(* CODESYS project tcl_stringutils.library
   Company: Red Rock Controls Limited
   Description: F_String_To_IPv4_Address added
   Version: 1.1.3.0
   Placeholder: tcl_StringUtils
   Author: Roger Christopher
   Title: tcl_StringUtils

Project tree, tasks and I/O mapping:
  libraries: Tc2_Standard, * (Beckhoff Automation GmbH); Tc2_System, * (Beckhoff Automation GmbH); Tc2_Utilities, * (Beckhoff Automation GmbH); Tc3_Module, * (Beckhoff Automation GmbH)
  Classes/
    function block T_LongString [ST]: AppendString, Clear, Address, Length
    function block T_StringSplitter [ST]: GetNext, GetRemainder, HasMore, Init
  Functions/
    Conversion/
      function F_String_To_IPv4_Address [ST]
      function F_TypeClassToString [ST]
      function F_ULINT_TO_TIMESTRUCT [ST]
    Date Time Formatting/
      function F_DateAsString [ST]
      function F_DateTimeAsString [ST]
      function F_DateTimeAsString_ms [ST]
      function F_TimeAsString [ST]
      function F_TimeAsString_ms [ST]
      function F_TimestampAsFilenameString [ST]
    String Formatting/
      function F_FormatString1 [ST]
      function F_FormatString10 [ST]
      function F_FormatString2 [ST]
      function F_FormatString3 [ST]
      function F_FormatString4 [ST]
      function F_FormatString5 [ST]
      function F_FormatString6 [ST]
      function F_FormatString7 [ST]
      function F_FormatString8 [ST]
      function F_FormatStringEx1 [ST]
      function F_FormatStringEx10 [ST]
      function F_FormatStringEx2 [ST]
      function F_FormatStringEx3 [ST]
      function F_FormatStringEx4 [ST]
      function F_FormatStringEx5 [ST]
      function F_FormatStringEx6 [ST]
      function F_FormatStringEx7 [ST]
      function F_FormatStringEx8 [ST]
      function F_LREAL_TO_STRING [ST]
      function F_LTrimEx [ST]
      function F_PadString [ST]
      function F_RTrimEx [ST]
      function F_STRING_TO_ARG [ST]
      function F_Trim [ST]
  Version/
    global variables Global_Version
  text list GlobalTextList
  global variables Param
*)

// Version/Global_Version
{attribute 'TcGenerated'}
{attribute 'no-analysis'}
{attribute 'linkalways'}
// This function has been automatically generated from the project information.
VAR_GLOBAL CONSTANT
	{attribute 'const_non_replaced'}
	stLibVersion_tcl_StringUtils : ST_LibVersion := (iMajor := 1, iMinor := 1, iBuild := 3, iRevision := 0, nFlags := 0, sVersion := '1.1.3.0');
END_VAR

// Param
{attribute 'qualified_only'}
VAR_GLOBAL CONSTANT
    MaxCsvFields : INT := 99;
END_VAR

// Classes/T_LongString
FUNCTION_BLOCK T_LongString
VAR
    buffer : STRING(MAX_LENGTH);
    CharCount : UDINT;
END_VAR
VAR CONSTANT
    MAX_LENGTH : UDINT := 1024;
END_VAR

METHOD AppendString
VAR_INPUT
    str : T_MaxString;
END_VAR
VAR
    stringLength : UDINT;
END_VAR
stringLength := INT_TO_UDINT(LEN(str));

IF (stringLength + CharCount < MAX_LENGTH - 1) THEN
    MEMCPY(
        destAddr := Address + CharCount,
        srcAddr  := ADR(str),
        n        := stringLength);
    CharCount := CharCount + stringLength;       
END_IF
END_METHOD

METHOD Clear
VAR_INPUT
END_VAR
MEMSET(Address,0,MAX_LENGTH);
CharCount := 0;
END_METHOD

PROPERTY Address : PVOID
GET
Address := ADR(Buffer);
END_GET
END_PROPERTY

PROPERTY Length : UDINT
GET
Length := CharCount;
END_GET
END_PROPERTY

END_FUNCTION_BLOCK

// Classes/T_StringSplitter
FUNCTION_BLOCK T_StringSplitter
VAR
	SubjectString : TC2_SYSTEM.T_MaxString;
	Delimiter : STRING;
	Delimiter1 : STRING;
	Delimiter2 : STRING;
	NextDelimiterPosition : INT;
	NextDelimiter1Position : INT;
	NextDelimiter2Position : INT;
END_VAR

METHOD GetNext : STRING(255)
VAR_INPUT
END_VAR
VAR
	RemainingLength: INT;
END_VAR
NextDelimiter1Position := FIND(SubjectString , Delimiter1);
NextDelimiter2Position := FIND(SubjectString , Delimiter2);

IF NextDelimiter1Position = 0 THEN
    // use Delimiter 2 position , even if zero...
    NextDelimiterPosition := NextDelimiter2Position;
    Delimiter := Delimiter2;
    
ELSIF NextDelimiter2Position = 0 THEN
    // use Delimiter 1 position , non-zero...
    NextDelimiterPosition := NextDelimiter1Position;
    Delimiter := Delimiter1;

ELSE
    // Both delimters found - use the one nearest the start of the string...
    IF NextDelimiter1Position < NextDelimiter2Position THEN
        NextDelimiterPosition := NextDelimiter1Position;
        Delimiter := Delimiter1;
    ELSE
        NextDelimiterPosition := NextDelimiter2Position;
        Delimiter := Delimiter2;
	END_IF
END_IF

IF NextDelimiterPosition > 0 THEN // delimitter found
    
    // extract next sub-string
	GetNext := LEFT(SubjectString,NextDelimiterPosition - 1);
    
    // remove sub-string from subject string
	RemainingLength := LEN(SubjectString) - NextDelimiterPosition - LEN(Delimiter) + 1;
	SubjectString := RIGHT(SubjectString,RemainingLength);
    
//    // strip any delimitters from front of remaining string
//    WHILE FIND(SubjectString,Delimiter1) = 1 DO
//        SubjectString := RIGHT(SubjectString,LEN(SubjectString) - LEN(Delimiter1));
//	END_WHILE
//    WHILE FIND(SubjectString,Delimiter2) = 1 DO
//        SubjectString := RIGHT(SubjectString,LEN(SubjectString) - LEN(Delimiter2));
//	END_WHILE
ELSE
	GetNext := SubjectString; // return what is left
	SubjectString := '';
END_IF
END_METHOD

METHOD GetRemainder : STRING(255)
GetRemainder := SubjectString; // return what is left
SubjectString := '';
END_METHOD

METHOD HasMore : BOOL
VAR_INPUT
END_VAR
HasMore := SubjectString <> '';
END_METHOD

METHOD Init
VAR_INPUT
		Str : TC2_SYSTEM.T_MaxString;
		Delim1 : STRING;
		Delim2 : STRING;
END_VAR
SubjectString := Str;
NextDelimiterPosition := 0;
Delimiter1 := Delim1;
Delimiter2 := Delim2;
END_METHOD

END_FUNCTION_BLOCK

// Functions/Conversion/F_String_To_IPv4_Address
FUNCTION F_String_To_IPv4_Address : ARRAY[1..4] of BYTE
VAR_INPUT
    IpAddress : STRING; // like 192.168.1.125
END_VAR
VAR
    StringSplitter : T_StringSplitter;
    Byte1          : STRING;
    Byte2          : STRING;
    Byte3          : STRING;
    Byte4          : STRING;
    Result         : ARRAY[1..4] OF BYTE;
END_VAR

StringSplitter.Init(IpAddress,
                    '.',
                    '');

Byte4 := StringSplitter.GetNext();
Byte3 := StringSplitter.GetNext();
Byte2 := StringSplitter.GetNext();
Byte1 := StringSplitter.GetNext();

Result[1] := STRING_TO_BYTE(Byte1);
Result[2] := STRING_TO_BYTE(Byte2);
Result[3] := STRING_TO_BYTE(Byte3);
Result[4] := STRING_TO_BYTE(Byte4);

F_String_To_IPv4_Address := Result;

END_FUNCTION

// Functions/Conversion/F_TypeClassToString
FUNCTION F_TypeClassToString : STRING
VAR_INPUT
    TypeClass : __SYSTEM.TYPE_CLASS;
END_VAR
VAR
    Result : STRING;
END_VAR

CASE TypeClass OF
    __SYSTEM.TYPE_CLASS.TYPE_BOOL          : Result := 'BOOL';
    __SYSTEM.TYPE_CLASS.TYPE_BIT           : Result := 'BOOL';
    __SYSTEM.TYPE_CLASS.TYPE_BYTE          : Result := 'BYTE';
    __SYSTEM.TYPE_CLASS.TYPE_WORD          : Result := 'WORD';
    __SYSTEM.TYPE_CLASS.TYPE_DWORD         : Result := 'DWORD';
    __SYSTEM.TYPE_CLASS.TYPE_LWORD         : Result := 'DWORD';
    __SYSTEM.TYPE_CLASS.TYPE_SINT          : Result := 'SINT';
    __SYSTEM.TYPE_CLASS.TYPE_INT           : Result := 'INT';
    __SYSTEM.TYPE_CLASS.TYPE_DINT          : Result := 'DINT';
    __SYSTEM.TYPE_CLASS.TYPE_LINT          : Result := 'LINT';
    __SYSTEM.TYPE_CLASS.TYPE_USINT         : Result := 'USINT';
    __SYSTEM.TYPE_CLASS.TYPE_UINT          : Result := 'UINT';
    __SYSTEM.TYPE_CLASS.TYPE_UDINT         : Result := 'UDINT';
    __SYSTEM.TYPE_CLASS.TYPE_ULINT         : Result := 'ULINT';
    __SYSTEM.TYPE_CLASS.TYPE_REAL          : Result := 'REAL';
    __SYSTEM.TYPE_CLASS.TYPE_LREAL         : Result := 'LREAL';
    __SYSTEM.TYPE_CLASS.TYPE_STRING        : Result := 'STRING';
    __SYSTEM.TYPE_CLASS.TYPE_WSTRING       : Result := 'WSTRING';     
    __SYSTEM.TYPE_CLASS.TYPE_TIME          : Result := 'TIME';        
    __SYSTEM.TYPE_CLASS.TYPE_DATE          : Result := 'DATE';        
    __SYSTEM.TYPE_CLASS.TYPE_DATEANDTIME   : Result := 'DATEANDTIME'; 
    __SYSTEM.TYPE_CLASS.TYPE_TIMEOFDAY     : Result := 'TIMEOFDAY';   
    __SYSTEM.TYPE_CLASS.TYPE_POINTER       : Result := 'POINTER';     
    __SYSTEM.TYPE_CLASS.TYPE_REFERENCE     : Result := 'REFERENCE';   
    __SYSTEM.TYPE_CLASS.TYPE_SUBRANGE      : Result := 'SUBRANGE';    
    __SYSTEM.TYPE_CLASS.TYPE_ENUM          : Result := 'ENUM';        
    __SYSTEM.TYPE_CLASS.TYPE_ARRAY         : Result := 'ARRAY';      
    __SYSTEM.TYPE_CLASS.TYPE_PARAMS        : Result := 'PARAMS';      
    __SYSTEM.TYPE_CLASS.TYPE_USERDEF       : Result := 'USERDEF';     
    __SYSTEM.TYPE_CLASS.TYPE_NONE          : Result := 'NONE';        
    __SYSTEM.TYPE_CLASS.TYPE_ANY           : Result := 'ANY';         
    __SYSTEM.TYPE_CLASS.TYPE_ANYBIT        : Result := 'ANYBIT';      
    __SYSTEM.TYPE_CLASS.TYPE_ANYDATE       : Result := 'ANYDATE';     
    __SYSTEM.TYPE_CLASS.TYPE_ANYINT        : Result := 'ANYINT';      
    __SYSTEM.TYPE_CLASS.TYPE_ANYNUM        : Result := 'ANYNUM';      
    __SYSTEM.TYPE_CLASS.TYPE_ANYREAL       : Result := 'ANYREAL';     
    __SYSTEM.TYPE_CLASS.TYPE_LAZY          : Result := 'LAZY';        
    __SYSTEM.TYPE_CLASS.TYPE_BITCONST      : Result := 'BITCONST';    
ELSE
    Result := DWORD_TO_STRING(TypeClass);
END_CASE

F_TypeClassToString := Result;

END_FUNCTION

// Functions/Conversion/F_ULINT_TO_TIMESTRUCT
FUNCTION F_ULINT_TO_TIMESTRUCT : TIMESTRUCT
VAR_INPUT
	TimeStamp : ULINT; // data type og eventLogger3 timestamp - number of 100nS since 1601
END_VAR
VAR
	pFileTime : POINTER TO T_FILETIME;
	Result : TIMESTRUCT;
END_VAR

pFileTime := ADR(TimeStamp);
Result := FILETIME_TO_SYSTEMTIME(pFileTime^);

F_ULINT_TO_TIMESTRUCT := Result;

END_FUNCTION

// Functions/Date Time Formatting/F_DateAsString
FUNCTION F_DateAsString : T_MaxString
VAR_INPUT
    TimeStruct : TIMESTRUCT;
END_VAR

F_DateAsString := F_FormatString3(
                      Format := '%.2d/%.2d/%.2d',
                      arg1   := F_WORD(TimeStruct.wDay),
                      arg2   := F_WORD(TimeStruct.wMonth),
                      arg3   := F_WORD(TimeStruct.wYear));

END_FUNCTION

// Functions/String Formatting/F_FormatString3
FUNCTION F_FormatString3 : T_MaxString
VAR_INPUT
	Format	: T_MaxString;
	arg1	: T_Arg;
	arg2	: T_Arg;
	arg3	: T_Arg;
END_VAR
VAR
    FB_FormatString1 : FB_FormatString;
END_VAR

FB_FormatString1(
	sFormat:= Format, 
	arg1:= arg1, 
	arg2:= arg2, 
	arg3:= arg3, 
	arg4:= , 
	arg5:= , 
	arg6:= , 
	arg7:= , 
	arg8:= , 
	arg9:= , 
	arg10:= , 
	bError=> , 
	nErrId=> , 
	sOut=> F_FormatString3);

END_FUNCTION

// Functions/Date Time Formatting/F_DateTimeAsString
FUNCTION F_DateTimeAsString : T_MaxString
VAR_INPUT
    TimeStruct : TIMESTRUCT;
END_VAR

F_DateTimeAsString := F_FormatStringEx2(
                          Format := '%s %s',
                          arg1   := F_TimeAsString(TimeStruct),
                          arg2   := F_DateAsString(TimeStruct));

END_FUNCTION

// Functions/String Formatting/F_FormatStringEx2
FUNCTION F_FormatStringEx2 : T_MaxString
VAR_INPUT
	Format	: T_MaxString;
	arg1	: T_MaxString;
	arg2	: T_MaxString;
END_VAR
VAR
    FB_FormatString1 : FB_FormatString;
END_VAR



FB_FormatString1(
	sFormat:= Format, 
	arg1:= F_STRING(arg1), 
	arg2:= F_STRING(arg2),
	arg3:= , 
	arg4:= , 
	arg5:= , 
	arg6:= , 
	arg7:= , 
	arg8:= , 
	arg9:= , 
	arg10:= , 
	bError=> , 
	nErrId=> , 
	sOut=> F_FormatStringEx2);

END_FUNCTION

// Functions/Date Time Formatting/F_TimeAsString
FUNCTION F_TimeAsString : T_MaxString
VAR_INPUT
    TimeStruct : TIMESTRUCT;
END_VAR

F_TimeAsString := F_FormatString3(
                      Format := '%.2d:%.2d:%.2d',
                      arg1   := F_WORD(TimeStruct.wHour),
                      arg2   := F_WORD(TimeStruct.wMinute),
                      arg3   := F_WORD(TimeStruct.wSecond));

END_FUNCTION

// Functions/Date Time Formatting/F_DateTimeAsString_ms
FUNCTION F_DateTimeAsString_ms : T_MaxString
VAR_INPUT
    TimeStruct : TIMESTRUCT;
END_VAR

F_DateTimeAsString_ms := F_FormatStringEx2(
                             Format := '%s %s',
                             arg1   := F_TimeAsString_ms(TimeStruct),
                             arg2   := F_DateAsString(TimeStruct));

END_FUNCTION

// Functions/Date Time Formatting/F_TimeAsString_ms
FUNCTION F_TimeAsString_ms : T_MaxString
VAR_INPUT
    TimeStruct : TIMESTRUCT;
END_VAR

F_TimeAsString_ms := F_FormatString4(
                         Format := '%.2d:%.2d:%.2d.%.3d',
                         arg1   := F_WORD(TimeStruct.wHour),
                         arg2   := F_WORD(TimeStruct.wMinute),
                         arg3   := F_WORD(TimeStruct.wSecond),
   	                     arg4   := F_WORD(TimeStruct.wMilliseconds));

END_FUNCTION

// Functions/String Formatting/F_FormatString4
FUNCTION F_FormatString4 : T_MaxString
VAR_INPUT
	Format	: T_MaxString;
	arg1	: T_Arg;
	arg2	: T_Arg;
	arg3	: T_Arg;
	arg4	: T_Arg;
END_VAR
VAR
    FB_FormatString1 : FB_FormatString;
END_VAR

FB_FormatString1(
	sFormat:= Format, 
	arg1:= arg1, 
	arg2:= arg2, 
	arg3:= arg3, 
	arg4:= arg4, 
	arg5:= , 
	arg6:= , 
	arg7:= , 
	arg8:= , 
	arg9:= , 
	arg10:= , 
	bError=> , 
	nErrId=> , 
	sOut=> F_FormatString4);

END_FUNCTION

// Functions/Date Time Formatting/F_TimestampAsFilenameString
FUNCTION F_TimestampAsFilenameString : T_MaxString
VAR_INPUT
    TimeStruct : TIMESTRUCT;
END_VAR
VAR
	FB_FormatString1 : FB_FormatString;
END_VAR

FB_FormatString1(
	sFormat:= '%.2d-%.2d-%.2d %.2d-%.2d-%.2d', 
	arg1:= F_WORD(TimeStruct.wYear), 
	arg2:= F_WORD(TimeStruct.wMonth), 
	arg3:= F_WORD(TimeStruct.wDay),
	arg4:= F_WORD(TimeStruct.wHour),
	arg5:= F_WORD(TimeStruct.wMinute), 
	arg6:= F_WORD(TimeStruct.wSecond), 
	arg7:= ,
	arg8:= , 
	arg9:= , 
	arg10:= , 
	bError=> , 
	nErrId=> , 
	sOut=> F_TimestampAsFilenameString);

END_FUNCTION

// Functions/String Formatting/F_FormatString1
FUNCTION F_FormatString1 : T_MaxString
VAR_INPUT
	Format	: T_MaxString;
	arg1	: T_Arg;
END_VAR
VAR
    FB_FormatString1 : FB_FormatString;
END_VAR

FB_FormatString1(
	sFormat:= Format, 
	arg1:= arg1, 
	arg2:= , 
	arg3:= , 
	arg4:= , 
	arg5:= , 
	arg6:= , 
	arg7:= , 
	arg8:= , 
	arg9:= , 
	arg10:= , 
	bError=> , 
	nErrId=> , 
	sOut=> F_FormatString1);

END_FUNCTION

// Functions/String Formatting/F_FormatString10
FUNCTION F_FormatString10 : T_MaxString
VAR_INPUT
	Format	: T_MaxString;
	arg1	: T_Arg;
	arg2	: T_Arg;
	arg3	: T_Arg;
	arg4	: T_Arg;
	arg5	: T_Arg;
	arg6	: T_Arg;
	arg7	: T_Arg;
	arg8	: T_Arg;
	arg9	: T_Arg;
	arg10	: T_Arg;
END_VAR
VAR
    FB_FormatString1 : FB_FormatString;
END_VAR

FB_FormatString1(
	sFormat:= Format, 
	arg1:= arg1, 
	arg2:= arg2, 
	arg3:= arg3, 
	arg4:= arg4, 
	arg5:= arg5, 
	arg6:= arg6, 
	arg7:= arg7, 
	arg8:= arg8, 
	arg9:= arg9, 
	arg10:= arg10, 
	bError=> , 
	nErrId=> , 
	sOut=> F_FormatString10);

END_FUNCTION

// Functions/String Formatting/F_FormatString2
FUNCTION F_FormatString2 : T_MaxString
VAR_INPUT
	Format	: T_MaxString;
	arg1	: T_Arg;
	arg2	: T_Arg;
END_VAR
VAR
    FB_FormatString1 : FB_FormatString;
END_VAR

FB_FormatString1(
	sFormat:= Format, 
	arg1:= arg1, 
	arg2:= arg2, 
	arg3:= , 
	arg4:= , 
	arg5:= , 
	arg6:= , 
	arg7:= , 
	arg8:= , 
	arg9:= , 
	arg10:= , 
	bError=> , 
	nErrId=> , 
	sOut=> F_FormatString2);

END_FUNCTION

// Functions/String Formatting/F_FormatString5
FUNCTION F_FormatString5 : T_MaxString
VAR_INPUT
	Format	: T_MaxString;
	arg1	: T_Arg;
	arg2	: T_Arg;
	arg3	: T_Arg;
	arg4	: T_Arg;
	arg5	: T_Arg;
END_VAR
VAR
    FB_FormatString1 : FB_FormatString;
END_VAR

FB_FormatString1(
	sFormat:= Format, 
	arg1:= arg1, 
	arg2:= arg2, 
	arg3:= arg3, 
	arg4:= arg4, 
	arg5:= arg5, 
	arg6:= , 
	arg7:= , 
	arg8:= , 
	arg9:= , 
	arg10:= , 
	bError=> , 
	nErrId=> , 
	sOut=> F_FormatString5);

END_FUNCTION

// Functions/String Formatting/F_FormatString6
FUNCTION F_FormatString6 : T_MaxString
VAR_INPUT
	Format	: T_MaxString;
	arg1	: T_Arg;
	arg2	: T_Arg;
	arg3	: T_Arg;
	arg4	: T_Arg;
	arg5	: T_Arg;
	arg6	: T_Arg;
END_VAR
VAR
    FB_FormatString1 : FB_FormatString;
END_VAR

FB_FormatString1(
	sFormat:= Format, 
	arg1:= arg1, 
	arg2:= arg2, 
	arg3:= arg3, 
	arg4:= arg4, 
	arg5:= arg5, 
	arg6:= arg6, 
	arg7:= , 
	arg8:= , 
	arg9:= , 
	arg10:= , 
	bError=> , 
	nErrId=> , 
	sOut=> F_FormatString6);

END_FUNCTION

// Functions/String Formatting/F_FormatString7
FUNCTION F_FormatString7 : T_MaxString
VAR_INPUT
	Format	: T_MaxString;
	arg1	: T_Arg;
	arg2	: T_Arg;
	arg3	: T_Arg;
	arg4	: T_Arg;
	arg5	: T_Arg;
	arg6	: T_Arg;
	arg7	: T_Arg;
END_VAR
VAR
    FB_FormatString1 : FB_FormatString;
END_VAR

FB_FormatString1(
	sFormat:= Format, 
	arg1:= arg1, 
	arg2:= arg2, 
	arg3:= arg3, 
	arg4:= arg4, 
	arg5:= arg5, 
	arg6:= arg6, 
	arg7:= arg7, 
	arg8:= , 
	arg9:= , 
	arg10:= , 
	bError=> , 
	nErrId=> , 
	sOut=> F_FormatString7);

END_FUNCTION

// Functions/String Formatting/F_FormatString8
FUNCTION F_FormatString8 : T_MaxString
VAR_INPUT
	Format	: T_MaxString;
	arg1	: T_Arg;
	arg2	: T_Arg;
	arg3	: T_Arg;
	arg4	: T_Arg;
	arg5	: T_Arg;
	arg6	: T_Arg;
	arg7	: T_Arg;
	arg8	: T_Arg;
END_VAR
VAR
    FB_FormatString1 : FB_FormatString;
END_VAR

FB_FormatString1(
	sFormat:= Format, 
	arg1:= arg1, 
	arg2:= arg2, 
	arg3:= arg3, 
	arg4:= arg4, 
	arg5:= arg5, 
	arg6:= arg6, 
	arg7:= arg7, 
	arg8:= arg8, 
	arg9:= , 
	arg10:= , 
	bError=> , 
	nErrId=> , 
	sOut=> F_FormatString8);

END_FUNCTION

// Functions/String Formatting/F_FormatStringEx1
FUNCTION F_FormatStringEx1 : T_MaxString
VAR_INPUT
	Format	: T_MaxString;
	arg1	: T_MaxString;
END_VAR
VAR
    FB_FormatString1 : FB_FormatString;
END_VAR



FB_FormatString1(
	sFormat:= Format, 
	arg1:= F_STRING(arg1), 
	arg2:= , 
	arg3:= , 
	arg4:= , 
	arg5:= , 
	arg6:= , 
	arg7:= , 
	arg8:= , 
	arg9:= , 
	arg10:= , 
	bError=> , 
	nErrId=> , 
	sOut=> F_FormatStringEx1);

END_FUNCTION

// Functions/String Formatting/F_FormatStringEx10
FUNCTION F_FormatStringEx10 : T_MaxString
VAR_INPUT
	Format	: T_MaxString;
	arg1	: T_MaxString;
	arg2	: T_MaxString;
	arg3	: T_MaxString;
	arg4	: T_MaxString;
	arg5	: T_MaxString;
	arg6	: T_MaxString;
	arg7	: T_MaxString;
	arg8	: T_MaxString;
	arg9	: T_MaxString;
	arg10	: T_MaxString;
END_VAR
VAR
    FB_FormatString1 : FB_FormatString;
END_VAR



FB_FormatString1(
	sFormat:= Format, 
	arg1 := F_STRING(arg1), 
	arg2 := F_STRING(arg2),
	arg3 := F_STRING(arg3), 
	arg4 := F_STRING(arg4), 
	arg5 := F_STRING(arg5), 
	arg6 := F_STRING(arg6), 
	arg7 := F_STRING(arg7), 
	arg8 := F_STRING(arg8),  
	arg9 := F_STRING(arg9), 
	arg10:= F_STRING(arg10), 
	bError=> , 
	nErrId=> , 
	sOut=> F_FormatStringEx10);

END_FUNCTION

// Functions/String Formatting/F_FormatStringEx3
FUNCTION F_FormatStringEx3 : T_MaxString
VAR_INPUT
	Format	: T_MaxString;
	arg1	: T_MaxString;
	arg2	: T_MaxString;
	arg3	: T_MaxString;
END_VAR
VAR
    FB_FormatString1 : FB_FormatString;
END_VAR



FB_FormatString1(
	sFormat:= Format, 
	arg1:= F_STRING(arg1), 
	arg2:= F_STRING(arg2),
	arg3:= F_STRING(arg3), 
	arg4:= , 
	arg5:= , 
	arg6:= , 
	arg7:= , 
	arg8:= , 
	arg9:= , 
	arg10:= , 
	bError=> , 
	nErrId=> , 
	sOut=> F_FormatStringEx3);

END_FUNCTION

// Functions/String Formatting/F_FormatStringEx4
FUNCTION F_FormatStringEx4 : T_MaxString
VAR_INPUT
	Format	: T_MaxString;
	arg1	: T_MaxString;
	arg2	: T_MaxString;
	arg3	: T_MaxString;
	arg4	: T_MaxString;
END_VAR
VAR
    FB_FormatString1 : FB_FormatString;
END_VAR



FB_FormatString1(
	sFormat:= Format, 
	arg1:= F_STRING(arg1), 
	arg2:= F_STRING(arg2),
	arg3:= F_STRING(arg3), 
	arg4:= F_STRING(arg4), 
	arg5:= , 
	arg6:= , 
	arg7:= , 
	arg8:= , 
	arg9:= , 
	arg10:= , 
	bError=> , 
	nErrId=> , 
	sOut=> F_FormatStringEx4);

END_FUNCTION

// Functions/String Formatting/F_FormatStringEx5
FUNCTION F_FormatStringEx5 : T_MaxString
VAR_INPUT
	Format	: T_MaxString;
	arg1	: T_MaxString;
	arg2	: T_MaxString;
	arg3	: T_MaxString;
	arg4	: T_MaxString;
	arg5	: T_MaxString;
END_VAR
VAR
    FB_FormatString1 : FB_FormatString;
END_VAR



FB_FormatString1(
	sFormat:= Format, 
	arg1:= F_STRING(arg1), 
	arg2:= F_STRING(arg2),
	arg3:= F_STRING(arg3), 
	arg4:= F_STRING(arg4), 
	arg5:= F_STRING(arg5), 
	arg6:= , 
	arg7:= , 
	arg8:= , 
	arg9:= , 
	arg10:= , 
	bError=> , 
	nErrId=> , 
	sOut=> F_FormatStringEx5);

END_FUNCTION

// Functions/String Formatting/F_FormatStringEx6
FUNCTION F_FormatStringEx6 : T_MaxString
VAR_INPUT
	Format	: T_MaxString;
	arg1	: T_MaxString;
	arg2	: T_MaxString;
	arg3	: T_MaxString;
	arg4	: T_MaxString;
	arg5	: T_MaxString;
	arg6	: T_MaxString;
END_VAR
VAR
    FB_FormatString1 : FB_FormatString;
END_VAR



FB_FormatString1(
	sFormat:= Format, 
	arg1:= F_STRING(arg1), 
	arg2:= F_STRING(arg2),
	arg3:= F_STRING(arg3), 
	arg4:= F_STRING(arg4), 
	arg5:= F_STRING(arg5), 
	arg6:= F_STRING(arg6), 
	arg7:= , 
	arg8:= , 
	arg9:= , 
	arg10:= , 
	bError=> , 
	nErrId=> , 
	sOut=> F_FormatStringEx6);

END_FUNCTION

// Functions/String Formatting/F_FormatStringEx7
FUNCTION F_FormatStringEx7 : T_MaxString
VAR_INPUT
	Format	: T_MaxString;
	arg1	: T_MaxString;
	arg2	: T_MaxString;
	arg3	: T_MaxString;
	arg4	: T_MaxString;
	arg5	: T_MaxString;
	arg6	: T_MaxString;
	arg7	: T_MaxString;
END_VAR
VAR
    FB_FormatString1 : FB_FormatString;
END_VAR



FB_FormatString1(
	sFormat:= Format, 
	arg1:= F_STRING(arg1), 
	arg2:= F_STRING(arg2),
	arg3:= F_STRING(arg3), 
	arg4:= F_STRING(arg4), 
	arg5:= F_STRING(arg5), 
	arg6:= F_STRING(arg6), 
	arg7:= F_STRING(arg7), 
	arg8:= ,  
	arg9:= , 
	arg10:= , 
	bError=> , 
	nErrId=> , 
	sOut=> F_FormatStringEx7);

END_FUNCTION

// Functions/String Formatting/F_FormatStringEx8
FUNCTION F_FormatStringEx8 : T_MaxString
VAR_INPUT
	Format	: T_MaxString;
	arg1	: T_MaxString;
	arg2	: T_MaxString;
	arg3	: T_MaxString;
	arg4	: T_MaxString;
	arg5	: T_MaxString;
	arg6	: T_MaxString;
	arg7	: T_MaxString;
	arg8	: T_MaxString;
END_VAR
VAR
    FB_FormatString1 : FB_FormatString;
END_VAR



FB_FormatString1(
	sFormat:= Format, 
	arg1:= F_STRING(arg1), 
	arg2:= F_STRING(arg2),
	arg3:= F_STRING(arg3), 
	arg4:= F_STRING(arg4), 
	arg5:= F_STRING(arg5), 
	arg6:= F_STRING(arg6), 
	arg7:= F_STRING(arg7), 
	arg8:= F_STRING(arg8),  
	arg9:= , 
	arg10:= , 
	bError=> , 
	nErrId=> , 
	sOut=> F_FormatStringEx8);

END_FUNCTION

// Functions/String Formatting/F_LREAL_TO_STRING
FUNCTION F_LREAL_TO_STRING : STRING
VAR_INPUT
    Value : LREAL;
    Precision : INT;
END_VAR
VAR
END_VAR

F_LREAL_TO_STRING := LREAL_TO_FMTSTR(in := Value,
                                     iPrecision := Precision,
                                     bRound := TRUE);

END_FUNCTION

// Functions/String Formatting/F_LTrimEx
FUNCTION F_LTrimEx : T_MaxString // removes n characters from start of string
VAR_INPUT
   n : UINT; 
   str : T_MaxString;
END_VAR
VAR
    Length : UINT;
END_VAR

Length := INT_TO_UINT(LEN(str));
IF n = 0 THEN
    F_LTrimEx := str;
ELSIF n < Length THEN
    MEMCPY(destAddr := ADR(F_LTrimEx),
           srcAddr  := ADR(str) + n,
           n        := Length - n + 1); // include null terminator
ELSE
	F_LTrimEx := ''; // remove everything
END_IF

END_FUNCTION

// Functions/String Formatting/F_PadString
FUNCTION F_PadString : T_MaxString // pad string with spaces or trim from rhs to fix length of string
VAR_INPUT
    InputString : T_MaxString;
    Length : UINT;
END_VAR
VAR
    InputStringLength : UINT;
    Result : T_MaxString;
    TrimLength : UINT;
    PaddingLength : UINT;
    i : UINT;
END_VAR

InputStringLength := INT_TO_UINT(MAX(0,LEN(InputString)));
Result := InputString;

IF InputStringLength > Length THEN
    TrimLength := InputStringLength - Length;
    Result := F_RTrimEx(TrimLength,Result);
    
ELSIF InputStringLength < Length THEN
    PaddingLength := Length - InputStringLength;

    FOR i := 1 TO PaddingLength DO
        Result := CONCAT(Result,' ');
	END_FOR
    
END_IF

F_PadString := Result;

END_FUNCTION

// Functions/String Formatting/F_RTrimEx
FUNCTION F_RTrimEx : T_MaxString // removes n characters from end of string
VAR_INPUT
   n : UINT; 
   str : T_MaxString;
END_VAR
VAR
    Length : UINT;
END_VAR

Length := INT_TO_UINT(LEN(str));
IF n = 0 THEN
    F_RTrimEx := str;
ELSIF n < Length THEN
    // overwrite chars to be trimmed with nulls...
    MEMSET(destAddr := ADR(str) + Length - n,
           fillByte:= 0,
           n := n); 
	F_RTrimEx := str;
ELSE
	F_RTrimEx := ''; // remove everything
END_IF

END_FUNCTION

// Functions/String Formatting/F_STRING_TO_ARG
FUNCTION F_STRING_TO_ARG : T_Arg
VAR_IN_OUT
    in : T_MaxString;
END_VAR
VAR
    Result : T_Arg;
END_VAR

Result.eType := E_ArgType.ARGTYPE_STRING;
Result.pData := ADR(in);
Result.cbLen := SIZEOF(in); // not LEN()! F_STRING gives LEN which does not work with CallRPC_Method args!

F_STRING_TO_ARG := Result;

END_FUNCTION

// Functions/String Formatting/F_Trim
FUNCTION F_Trim : T_MaxString
VAR_INPUT
	str: T_MaxString;
END_VAR
VAR
	Result: T_MaxString;
END_VAR

Result := str;
WHILE 
    LEFT(Result,1) = '$T'
OR 
    LEFT(Result,1) = ' '
DO
	Result := F_LTrimEx(n := 1, str := Result); // Strip tabs and spaces from LHS
END_WHILE

WHILE 
    RIGHT(Result,1) = '$R'
OR 
    RIGHT(Result,1) = '$N'
OR 
    RIGHT(Result,1) = '$T'
OR 
    RIGHT(Result,1) = ' '
DO
	Result := F_RTrimEx(n := 1, str := Result); // Strip tabs, Spaces, CR and LF from RHS
END_WHILE


F_Trim := Result;

END_FUNCTION
